{attribute 'GeneratedUsingTerminal: EJ7211-0010-0030'}
{attribute addProperty BoxType "EJ7211-0010-0030"}
{attribute addProperty Id "AdsAddrAT %I*.TcoAmsAddr0DcOutputShiftAT %I*DINT4DcInputShiftAT %I*DINT4Chn0AT %I*USINT1Chn1AT %I*USINT1StateAT %I*UINT2"}
{attribute addProperty CRC "258765876"}
{attribute addProperty Size "12"}
TYPE InfoData_0F6C7434 EXTENDS InputBase_8311D824 :
STRUCT
	{attribute addProperty Name "AdsAddr"}
	AdsAddr AT %I* : .TcoAmsAddr;
	{attribute addProperty Name "DcOutputShift"}
	DcOutputShift AT %I* : DINT;
	{attribute addProperty Name "DcInputShift"}
	DcInputShift AT %I* : DINT;
	{attribute addProperty Name "Chn0"}
	Chn0 AT %I* : USINT;
	{attribute addProperty Name "Chn1"}
	Chn1 AT %I* : USINT;
	{attribute addProperty Name "State"}
	State AT %I* : UINT;
END_STRUCT
END_TYPE

(* stored: Version 1.2.0.0, ProductVersion 3.1.4024.9
   DUT InfoData_0F6C7434: Id {6933ca41-1c5a-47fd-a2ac-2185840a6668} *)
